(*program for setting parameters for FileOpenSae visualization dialog*)
PROGRAM P_FileDialog
VAR
	fbFileList                              : Visu_FbFileListProvider; 
	sSelectedDirectory						: STRING;
	sSelectedFileName						: STRING;
	iCount									: INT;
	bOpen 									: BOOL;
	sDir									: STRING(255):='C:\';
	bFile									: BOOL:=TRUE;
END_VAR

IF bFile OR bOpen THEN
	fbFileList.Initialize(
                        stDirectory:= sDir, 
                        stFilter:='Text Files(*.txt)|*.txt' , 
                        stFileIn:='', 
                        stTitle:= 'Dialog file open', 
                        iRowCount:=10 , 
                        bBrowseDirectory:= TRUE, 
                        bTouch:=FALSE ); 
	bFile:=FALSE;
END_IF
					
 
sSelectedDirectory:=fbFileList.GetSelectedDirectory();
sSelectedFileName:=fbFileList.GetSelectedFileName();
iCount:=fbFileList.Count;

END_PROGRAM

(* stored: Version 1.1.0.1, ProductVersion 3.1.4024.3
   POU P_FileDialog: Id {f070ba40-c611-4c81-984d-b38cc80f04b9}, SpecialFunc None *)
